Universal Robots PolyScope program: rtde_control_loop.urp

Program rtde_control_loop (installation=default directory=/ursim/programs/rtde-2.4.8/examples createdIn=5.4.2.76197 lastSavedIn=5.4.2.76197 robotSerialNumber=20183099999)
Calibrated DH parameters: a=[0, -0.6127, -0.57155, 0, 0, 0]; d=[0.1807, 0, 0, 0.17415, 0.11985, 0.11655]; alpha=[1.570796, 0, 0, 1.570796, -1.570796, 0]; deltaTheta=[0, 0, 0, 0, 0, 0]
Robot Program (runOnlyOnce=false)
  MoveP speed 250 mm/s, acceleration 1200 mm/s^2 (blendRadius=0.025 useActiveTCP=true) feature=Base
    Waypoint Waypoint_1: TCP in base x=-189.632 y=-609.684 z=260.971 mm, rx=-0.0012 ry=3.1163 rz=0.0389 rad; joints [-91.713, -98.956, -126.223, -46.295, 91.392, -1.776] deg
